(* CODESYS project Estação 2 - Measuring (2022).project

Project tree, tasks and I/O mapping:
  Device : CPX-CEC-C1-V3, Festo AG & Co. KG, order no. 3473128, version 3.5.7.37
      unmapped channels: Rotary switch
    application Application
      libraries: Standard, * (System); CAA CiA 405, 3.5.7.0 (CAA Technical Workgroup)
      task MainTask (cyclic, interval t#20ms, priority 20) calls PLC_PRG
      program PLC_PRG [ST]
      function ATUALIZAR_VALORES [ST]
      visualisation Visualization
      global variables GVL
      function INICIALIZACAO [ST]
      program teste_comunicacao [ST]
    CANbus : CANbus, 3S - Smart Software Solutions GmbH, version 3.5.12.0
        settings: Baudrate = 1000 kbit/s
      CANopen_Manager : CANopen_Manager, 3S - Smart Software Solutions GmbH, version 3.5.10.0
          settings: Sync CycleTime in Microseconds = 8000; Synchronous Window Length = 0; Enable Heartbeat generation = FALSE; Factory Settings Default = FALSE; Expert Settings Default = TRUE; ConfigVersion = 50659584
        CTEU_CO : CTEU-CO, Festo AG & Co. KG, order no. 570038, version 0.3223089.CTEU_CO.3.3
            settings: NODEIDSAVED = 1; SDO Timeout = 1000000; EXPERTSETTINGS = TRUE; PDO 16#1400.COBID = 16#00000201; Process by CANopenManager = TRUE; PDO 16#1401.COBID = 16#00000301; Process by CANopenManager = TRUE; PDO 16#1800.COBID = 16#00000181; Process by CANopenManager = TRUE; PDO 16#1801.COBID = 16#00000281; Process by CANopenManager = TRUE; 8-Bit Digital Output 1-8.Subindex = 16#01; 8-Bit Digital Output 9-16.Subindex = 16#02; 8-Bit Digital Output 17-24.Subindex = 16#03; 8-Bit Digital Output 25-32.Subindex = 16#04; 8-Bit Digital Output 33-40.Subindex = 16#05; 8-Bit Digital Output 41-48.Subindex = 16#06; 8-Bit Digital Output 49-56.Subindex = 16#07; 8-Bit Digital Output 75-64.Subindex = 16#08; 8-Bit Digital Output 65-72.Subindex = 16#09; 8-Bit Digital Output 73-80.Subindex = 16#0A; 8-Bit Digital Output 81-88.Subindex = 16#0B; 8-Bit Digital Output 89-96.Subindex = 16#0C; 8-Bit Digital Output 97-104.Subindex = 16#0D; 8-Bit Digital Output 105-112.Subindex = 16#0E; 8-Bit Digital Output 113-120.Subindex = 16#0F; 8-Bit Digital Input 1-8.Subindex = 16#01; 8-Bit Digital Input 9-16.Subindex = 16#02; 8-Bit Digital Input 17-24.Subindex = 16#03; 8-Bit Digital Input 25-32.Subindex = 16#04; 8-Bit Digital Input 33-40.Subindex = 16#05; 8-Bit Digital Input 41-48.Subindex = 16#06; 8-Bit Digital Input 49-56.Subindex = 16#07; 8-Bit Digital Input 57-64.Subindex = 16#08; 8-Bit Digital Input 65-72.Subindex = 16#09; 8-Bit Digital Input 73-80.Subindex = 16#0A; 8-Bit Digital Input 81-88.Subindex = 16#0B; 8-Bit Digital Input 89-96.Subindex = 16#0C; 8-Bit Digital Input 97-104.Subindex = 16#0D; 8-Bit Digital Input 105-112.Subindex = 16#0E;
              8-Bit Digital Input 113-120.Subindex = 16#0F; SDO List.Set Guardtime.Index = 16#100C; SDO List.Set Guardtime.Subindex = 16#00; SDO List.Set Guardtime.Value = 16#00000000; SDO List.Set Guardtime.Size = 16; SDO List.Set Guardtime.AbortIfError = FALSE; SDO List.Set Guardtime.JumpToLine = FALSE; SDO List.Set Guardtime.Line = 0; SDO List.Set Lifetime.Index = 16#100D; SDO List.Set Lifetime.Subindex = 16#00; SDO List.Set Lifetime.Value = 16#00000000; SDO List.Set Lifetime.Size = 8; SDO List.Set Lifetime.AbortIfError = FALSE; SDO List.Set Lifetime.JumpToLine = FALSE; SDO List.Set Lifetime.Line = 0; SDO List.Set Heartbeat Consumer.Index = 16#1016; SDO List.Set Heartbeat Consumer.Subindex = 16#01; SDO List.Set Heartbeat Consumer.Value = 0; SDO List.Set Heartbeat Consumer.Size = 32; SDO List.Set Heartbeat Consumer.AbortIfError = FALSE; SDO List.Set Heartbeat Consumer.JumpToLine = FALSE; SDO List.Set Heartbeat Consumer.Line = 0; SDO List.Set Heartbeat Consumer.Index = 16#1016; SDO List.Set Heartbeat Consumer.Subindex = 16#02; SDO List.Set Heartbeat Consumer.Value = 0; SDO List.Set Heartbeat Consumer.Size = 32; SDO List.Set Heartbeat Consumer.AbortIfError = FALSE; SDO List.Set Heartbeat Consumer.JumpToLine = FALSE; SDO List.Set Heartbeat Consumer.Line = 0; SDO List.Set Heartbeat Consumer.Index = 16#1016; SDO List.Set Heartbeat Consumer.Subindex = 16#03; SDO List.Set Heartbeat Consumer.Value = 0; SDO List.Set Heartbeat Consumer.Size = 32; SDO List.Set Heartbeat Consumer.AbortIfError = FALSE; SDO List.Set Heartbeat Consumer.JumpToLine = FALSE; SDO List.Set Heartbeat Consumer.Line = 0; SDO List.Set Heartbeat Producer.Index = 16#1017; SDO List.Set Heartbeat Producer.Subindex = 16#00; SDO List.Set Heartbeat Producer.Value = 16#00000000; SDO List.Set Heartbeat Producer.Size = 16;
              SDO List.Set Heartbeat Producer.AbortIfError = FALSE; SDO List.Set Heartbeat Producer.JumpToLine = FALSE; SDO List.Set Heartbeat Producer.Line = 0; SDO List.Disable PDO.Index = 16#1400; SDO List.Disable PDO.Subindex = 16#01; SDO List.Disable PDO.Value = 16#80000201; SDO List.Disable PDO.Size = 32; SDO List.Disable PDO.AbortIfError = FALSE; SDO List.Disable PDO.JumpToLine = FALSE; SDO List.Disable PDO.Line = 0; SDO List.Set transmission type.Index = 16#1400; SDO List.Set transmission type.Subindex = 16#02; SDO List.Set transmission type.Value = 16#FF; SDO List.Set transmission type.Size = 8; SDO List.Set transmission type.AbortIfError = FALSE; SDO List.Set transmission type.JumpToLine = FALSE; SDO List.Set transmission type.Line = 0; SDO List.Clear pdo mapping.Index = 16#1600; SDO List.Clear pdo mapping.Subindex = 16#00; SDO List.Clear pdo mapping.Value = 16#0; SDO List.Clear pdo mapping.Size = 8; SDO List.Clear pdo mapping.AbortIfError = FALSE; SDO List.Clear pdo mapping.JumpToLine = FALSE; SDO List.Clear pdo mapping.Line = 0; SDO List.Set Mapping.Index = 16#1600; SDO List.Set Mapping.Subindex = 16#01; SDO List.Set Mapping.Value = 16#62000108; SDO List.Set Mapping.Size = 32; SDO List.Set Mapping.AbortIfError = FALSE; SDO List.Set Mapping.JumpToLine = FALSE; SDO List.Set Mapping.Line = 0; SDO List.Set Mapping.Index = 16#1600; SDO List.Set Mapping.Subindex = 16#02; SDO List.Set Mapping.Value = 16#62000208; SDO List.Set Mapping.Size = 32; SDO List.Set Mapping.AbortIfError = FALSE; SDO List.Set Mapping.JumpToLine = FALSE; SDO List.Set Mapping.Line = 0; SDO List.Set Mapping.Index = 16#1600; SDO List.Set Mapping.Subindex = 16#03;
              SDO List.Set Mapping.Value = 16#62000308; SDO List.Set Mapping.Size = 32; SDO List.Set Mapping.AbortIfError = FALSE; SDO List.Set Mapping.JumpToLine = FALSE; SDO List.Set Mapping.Line = 0; SDO List.Set Mapping.Index = 16#1600; SDO List.Set Mapping.Subindex = 16#04; SDO List.Set Mapping.Value = 16#62000408; SDO List.Set Mapping.Size = 32; SDO List.Set Mapping.AbortIfError = FALSE; SDO List.Set Mapping.JumpToLine = FALSE; SDO List.Set Mapping.Line = 0; SDO List.Set Mapping.Index = 16#1600; SDO List.Set Mapping.Subindex = 16#05; SDO List.Set Mapping.Value = 16#62000508; SDO List.Set Mapping.Size = 32; SDO List.Set Mapping.AbortIfError = FALSE; SDO List.Set Mapping.JumpToLine = FALSE; SDO List.Set Mapping.Line = 0; SDO List.Set Mapping.Index = 16#1600; SDO List.Set Mapping.Subindex = 16#06; SDO List.Set Mapping.Value = 16#62000608; SDO List.Set Mapping.Size = 32; SDO List.Set Mapping.AbortIfError = FALSE; SDO List.Set Mapping.JumpToLine = FALSE; SDO List.Set Mapping.Line = 0; SDO List.Set Mapping.Index = 16#1600; SDO List.Set Mapping.Subindex = 16#07; SDO List.Set Mapping.Value = 16#62000708; SDO List.Set Mapping.Size = 32; SDO List.Set Mapping.AbortIfError = FALSE; SDO List.Set Mapping.JumpToLine = FALSE; SDO List.Set Mapping.Line = 0; SDO List.Set Mapping.Index = 16#1600; SDO List.Set Mapping.Subindex = 16#08; SDO List.Set Mapping.Value = 16#62000808; SDO List.Set Mapping.Size = 32; SDO List.Set Mapping.AbortIfError = FALSE; SDO List.Set Mapping.JumpToLine = FALSE; SDO List.Set Mapping.Line = 0;
              SDO List.Set number of mappings.Index = 16#1600; SDO List.Set number of mappings.Subindex = 16#00; SDO List.Set number of mappings.Value = 16#08; SDO List.Set number of mappings.Size = 8; SDO List.Set number of mappings.AbortIfError = FALSE; SDO List.Set number of mappings.JumpToLine = FALSE; SDO List.Set number of mappings.Line = 0; SDO List.Set and enable COB-ID.Index = 16#1400; SDO List.Set and enable COB-ID.Subindex = 16#01; SDO List.Set and enable COB-ID.Value = 16#00000201; SDO List.Set and enable COB-ID.Size = 32; SDO List.Set and enable COB-ID.AbortIfError = FALSE; SDO List.Set and enable COB-ID.JumpToLine = FALSE; SDO List.Set and enable COB-ID.Line = 0; SDO List.Disable PDO.Index = 16#1401; SDO List.Disable PDO.Subindex = 16#01; SDO List.Disable PDO.Value = 16#80000301; SDO List.Disable PDO.Size = 32; SDO List.Disable PDO.AbortIfError = FALSE; SDO List.Disable PDO.JumpToLine = FALSE; SDO List.Disable PDO.Line = 0; SDO List.Set transmission type.Index = 16#1401; SDO List.Set transmission type.Subindex = 16#02; SDO List.Set transmission type.Value = 16#FF; SDO List.Set transmission type.Size = 8; SDO List.Set transmission type.AbortIfError = FALSE; SDO List.Set transmission type.JumpToLine = FALSE; SDO List.Set transmission type.Line = 0; SDO List.Clear pdo mapping.Index = 16#1601; SDO List.Clear pdo mapping.Subindex = 16#00; SDO List.Clear pdo mapping.Value = 16#0; SDO List.Clear pdo mapping.Size = 8; SDO List.Clear pdo mapping.AbortIfError = FALSE; SDO List.Clear pdo mapping.JumpToLine = FALSE; SDO List.Clear pdo mapping.Line = 0; SDO List.Set Mapping.Index = 16#1601; SDO List.Set Mapping.Subindex = 16#01; SDO List.Set Mapping.Value = 16#62000908; SDO List.Set Mapping.Size = 32; SDO List.Set Mapping.AbortIfError = FALSE;
              SDO List.Set Mapping.JumpToLine = FALSE; SDO List.Set Mapping.Line = 0; SDO List.Set Mapping.Index = 16#1601; SDO List.Set Mapping.Subindex = 16#02; SDO List.Set Mapping.Value = 16#62000A08; SDO List.Set Mapping.Size = 32; SDO List.Set Mapping.AbortIfError = FALSE; SDO List.Set Mapping.JumpToLine = FALSE; SDO List.Set Mapping.Line = 0; SDO List.Set Mapping.Index = 16#1601; SDO List.Set Mapping.Subindex = 16#03; SDO List.Set Mapping.Value = 16#62000B08; SDO List.Set Mapping.Size = 32; SDO List.Set Mapping.AbortIfError = FALSE; SDO List.Set Mapping.JumpToLine = FALSE; SDO List.Set Mapping.Line = 0; SDO List.Set Mapping.Index = 16#1601; SDO List.Set Mapping.Subindex = 16#04; SDO List.Set Mapping.Value = 16#62000C08; SDO List.Set Mapping.Size = 32; SDO List.Set Mapping.AbortIfError = FALSE; SDO List.Set Mapping.JumpToLine = FALSE; SDO List.Set Mapping.Line = 0; SDO List.Set Mapping.Index = 16#1601; SDO List.Set Mapping.Subindex = 16#05; SDO List.Set Mapping.Value = 16#62000D08; SDO List.Set Mapping.Size = 32; SDO List.Set Mapping.AbortIfError = FALSE; SDO List.Set Mapping.JumpToLine = FALSE; SDO List.Set Mapping.Line = 0; SDO List.Set Mapping.Index = 16#1601; SDO List.Set Mapping.Subindex = 16#06; SDO List.Set Mapping.Value = 16#62000E08; SDO List.Set Mapping.Size = 32; SDO List.Set Mapping.AbortIfError = FALSE; SDO List.Set Mapping.JumpToLine = FALSE; SDO List.Set Mapping.Line = 0; SDO List.Set Mapping.Index = 16#1601; SDO List.Set Mapping.Subindex = 16#07; SDO List.Set Mapping.Value = 16#62000F08;
              SDO List.Set Mapping.Size = 32; SDO List.Set Mapping.AbortIfError = FALSE; SDO List.Set Mapping.JumpToLine = FALSE; SDO List.Set Mapping.Line = 0; SDO List.Set Mapping.Index = 16#1601; SDO List.Set Mapping.Subindex = 16#08; SDO List.Set Mapping.Value = 16#62001008; SDO List.Set Mapping.Size = 32; SDO List.Set Mapping.AbortIfError = FALSE; SDO List.Set Mapping.JumpToLine = FALSE; SDO List.Set Mapping.Line = 0; SDO List.Set number of mappings.Index = 16#1601; SDO List.Set number of mappings.Subindex = 16#00; SDO List.Set number of mappings.Value = 16#08; SDO List.Set number of mappings.Size = 8; SDO List.Set number of mappings.AbortIfError = FALSE; SDO List.Set number of mappings.JumpToLine = FALSE; SDO List.Set number of mappings.Line = 0; SDO List.Set and enable COB-ID.Index = 16#1401; SDO List.Set and enable COB-ID.Subindex = 16#01; SDO List.Set and enable COB-ID.Value = 16#00000301; SDO List.Set and enable COB-ID.Size = 32; SDO List.Set and enable COB-ID.AbortIfError = FALSE; SDO List.Set and enable COB-ID.JumpToLine = FALSE; SDO List.Set and enable COB-ID.Line = 0; SDO List.Disable PDO.Index = 16#1800; SDO List.Disable PDO.Subindex = 16#01; SDO List.Disable PDO.Value = 16#80000181; SDO List.Disable PDO.Size = 32; SDO List.Disable PDO.AbortIfError = FALSE; SDO List.Disable PDO.JumpToLine = FALSE; SDO List.Disable PDO.Line = 0; SDO List.Set transmission type.Index = 16#1800; SDO List.Set transmission type.Subindex = 16#02; SDO List.Set transmission type.Value = 16#FF; SDO List.Set transmission type.Size = 8; SDO List.Set transmission type.AbortIfError = FALSE; SDO List.Set transmission type.JumpToLine = FALSE; SDO List.Set transmission type.Line = 0; SDO List.Set inhibit time.Index = 16#1800;
              SDO List.Set inhibit time.Subindex = 16#03; SDO List.Set inhibit time.Value = 16#0000; SDO List.Set inhibit time.Size = 16; SDO List.Set inhibit time.AbortIfError = FALSE; SDO List.Set inhibit time.JumpToLine = FALSE; SDO List.Set inhibit time.Line = 0; SDO List.Set event time.Index = 16#1800; SDO List.Set event time.Subindex = 16#05; SDO List.Set event time.Value = 16#0000; SDO List.Set event time.Size = 16; SDO List.Set event time.AbortIfError = FALSE; SDO List.Set event time.JumpToLine = FALSE; SDO List.Set event time.Line = 0; SDO List.Clear pdo mapping.Index = 16#1A00; SDO List.Clear pdo mapping.Subindex = 16#00; SDO List.Clear pdo mapping.Value = 16#0; SDO List.Clear pdo mapping.Size = 8; SDO List.Clear pdo mapping.AbortIfError = FALSE; SDO List.Clear pdo mapping.JumpToLine = FALSE; SDO List.Clear pdo mapping.Line = 0; SDO List.Set Mapping.Index = 16#1A00; SDO List.Set Mapping.Subindex = 16#01; SDO List.Set Mapping.Value = 16#60000108; SDO List.Set Mapping.Size = 32; SDO List.Set Mapping.AbortIfError = FALSE; SDO List.Set Mapping.JumpToLine = FALSE; SDO List.Set Mapping.Line = 0; SDO List.Set Mapping.Index = 16#1A00; SDO List.Set Mapping.Subindex = 16#02; SDO List.Set Mapping.Value = 16#60000208; SDO List.Set Mapping.Size = 32; SDO List.Set Mapping.AbortIfError = FALSE; SDO List.Set Mapping.JumpToLine = FALSE; SDO List.Set Mapping.Line = 0; SDO List.Set Mapping.Index = 16#1A00; SDO List.Set Mapping.Subindex = 16#03; SDO List.Set Mapping.Value = 16#60000308; SDO List.Set Mapping.Size = 32; SDO List.Set Mapping.AbortIfError = FALSE; SDO List.Set Mapping.JumpToLine = FALSE;
              SDO List.Set Mapping.Line = 0; SDO List.Set Mapping.Index = 16#1A00; SDO List.Set Mapping.Subindex = 16#04; SDO List.Set Mapping.Value = 16#60000408; SDO List.Set Mapping.Size = 32; SDO List.Set Mapping.AbortIfError = FALSE; SDO List.Set Mapping.JumpToLine = FALSE; SDO List.Set Mapping.Line = 0; SDO List.Set Mapping.Index = 16#1A00; SDO List.Set Mapping.Subindex = 16#05; SDO List.Set Mapping.Value = 16#60000508; SDO List.Set Mapping.Size = 32; SDO List.Set Mapping.AbortIfError = FALSE; SDO List.Set Mapping.JumpToLine = FALSE; SDO List.Set Mapping.Line = 0; SDO List.Set Mapping.Index = 16#1A00; SDO List.Set Mapping.Subindex = 16#06; SDO List.Set Mapping.Value = 16#60000608; SDO List.Set Mapping.Size = 32; SDO List.Set Mapping.AbortIfError = FALSE; SDO List.Set Mapping.JumpToLine = FALSE; SDO List.Set Mapping.Line = 0; SDO List.Set Mapping.Index = 16#1A00; SDO List.Set Mapping.Subindex = 16#07; SDO List.Set Mapping.Value = 16#60000708; SDO List.Set Mapping.Size = 32; SDO List.Set Mapping.AbortIfError = FALSE; SDO List.Set Mapping.JumpToLine = FALSE; SDO List.Set Mapping.Line = 0; SDO List.Set Mapping.Index = 16#1A00; SDO List.Set Mapping.Subindex = 16#08; SDO List.Set Mapping.Value = 16#60000808; SDO List.Set Mapping.Size = 32; SDO List.Set Mapping.AbortIfError = FALSE; SDO List.Set Mapping.JumpToLine = FALSE; SDO List.Set Mapping.Line = 0; SDO List.Set number of mappings.Index = 16#1A00; SDO List.Set number of mappings.Subindex = 16#00; SDO List.Set number of mappings.Value = 16#08; SDO List.Set number of mappings.Size = 8;
              SDO List.Set number of mappings.AbortIfError = FALSE; SDO List.Set number of mappings.JumpToLine = FALSE; SDO List.Set number of mappings.Line = 0; SDO List.Set and enable COB-ID.Index = 16#1800; SDO List.Set and enable COB-ID.Subindex = 16#01; SDO List.Set and enable COB-ID.Value = 16#00000181; SDO List.Set and enable COB-ID.Size = 32; SDO List.Set and enable COB-ID.AbortIfError = FALSE; SDO List.Set and enable COB-ID.JumpToLine = FALSE; SDO List.Set and enable COB-ID.Line = 0; SDO List.Disable PDO.Index = 16#1801; SDO List.Disable PDO.Subindex = 16#01; SDO List.Disable PDO.Value = 16#80000281; SDO List.Disable PDO.Size = 32; SDO List.Disable PDO.AbortIfError = FALSE; SDO List.Disable PDO.JumpToLine = FALSE; SDO List.Disable PDO.Line = 0; SDO List.Set transmission type.Index = 16#1801; SDO List.Set transmission type.Subindex = 16#02; SDO List.Set transmission type.Value = 16#FF; SDO List.Set transmission type.Size = 8; SDO List.Set transmission type.AbortIfError = FALSE; SDO List.Set transmission type.JumpToLine = FALSE; SDO List.Set transmission type.Line = 0; SDO List.Set inhibit time.Index = 16#1801; SDO List.Set inhibit time.Subindex = 16#03; SDO List.Set inhibit time.Value = 16#0000; SDO List.Set inhibit time.Size = 16; SDO List.Set inhibit time.AbortIfError = FALSE; SDO List.Set inhibit time.JumpToLine = FALSE; SDO List.Set inhibit time.Line = 0; SDO List.Set event time.Index = 16#1801; SDO List.Set event time.Subindex = 16#05; SDO List.Set event time.Value = 16#0000; SDO List.Set event time.Size = 16; SDO List.Set event time.AbortIfError = FALSE; SDO List.Set event time.JumpToLine = FALSE; SDO List.Set event time.Line = 0; SDO List.Clear pdo mapping.Index = 16#1A01; SDO List.Clear pdo mapping.Subindex = 16#00;
              SDO List.Clear pdo mapping.Value = 16#0; SDO List.Clear pdo mapping.Size = 8; SDO List.Clear pdo mapping.AbortIfError = FALSE; SDO List.Clear pdo mapping.JumpToLine = FALSE; SDO List.Clear pdo mapping.Line = 0; SDO List.Set Mapping.Index = 16#1A01; SDO List.Set Mapping.Subindex = 16#01; SDO List.Set Mapping.Value = 16#60000908; SDO List.Set Mapping.Size = 32; SDO List.Set Mapping.AbortIfError = FALSE; SDO List.Set Mapping.JumpToLine = FALSE; SDO List.Set Mapping.Line = 0; SDO List.Set Mapping.Index = 16#1A01; SDO List.Set Mapping.Subindex = 16#02; SDO List.Set Mapping.Value = 16#60000A08; SDO List.Set Mapping.Size = 32; SDO List.Set Mapping.AbortIfError = FALSE; SDO List.Set Mapping.JumpToLine = FALSE; SDO List.Set Mapping.Line = 0; SDO List.Set Mapping.Index = 16#1A01; SDO List.Set Mapping.Subindex = 16#03; SDO List.Set Mapping.Value = 16#60000B08; SDO List.Set Mapping.Size = 32; SDO List.Set Mapping.AbortIfError = FALSE; SDO List.Set Mapping.JumpToLine = FALSE; SDO List.Set Mapping.Line = 0; SDO List.Set Mapping.Index = 16#1A01; SDO List.Set Mapping.Subindex = 16#04; SDO List.Set Mapping.Value = 16#60000C08; SDO List.Set Mapping.Size = 32; SDO List.Set Mapping.AbortIfError = FALSE; SDO List.Set Mapping.JumpToLine = FALSE; SDO List.Set Mapping.Line = 0; SDO List.Set Mapping.Index = 16#1A01; SDO List.Set Mapping.Subindex = 16#05; SDO List.Set Mapping.Value = 16#60000D08; SDO List.Set Mapping.Size = 32; SDO List.Set Mapping.AbortIfError = FALSE; SDO List.Set Mapping.JumpToLine = FALSE; SDO List.Set Mapping.Line = 0;
              SDO List.Set Mapping.Index = 16#1A01; SDO List.Set Mapping.Subindex = 16#06; SDO List.Set Mapping.Value = 16#60000E08; SDO List.Set Mapping.Size = 32; SDO List.Set Mapping.AbortIfError = FALSE; SDO List.Set Mapping.JumpToLine = FALSE; SDO List.Set Mapping.Line = 0; SDO List.Set Mapping.Index = 16#1A01; SDO List.Set Mapping.Subindex = 16#07; SDO List.Set Mapping.Value = 16#60000F08; SDO List.Set Mapping.Size = 32; SDO List.Set Mapping.AbortIfError = FALSE; SDO List.Set Mapping.JumpToLine = FALSE; SDO List.Set Mapping.Line = 0; SDO List.Set Mapping.Index = 16#1A01; SDO List.Set Mapping.Subindex = 16#08; SDO List.Set Mapping.Value = 16#60001008; SDO List.Set Mapping.Size = 32; SDO List.Set Mapping.AbortIfError = FALSE; SDO List.Set Mapping.JumpToLine = FALSE; SDO List.Set Mapping.Line = 0; SDO List.Set number of mappings.Index = 16#1A01; SDO List.Set number of mappings.Subindex = 16#00; SDO List.Set number of mappings.Value = 16#08; SDO List.Set number of mappings.Size = 8; SDO List.Set number of mappings.AbortIfError = FALSE; SDO List.Set number of mappings.JumpToLine = FALSE; SDO List.Set number of mappings.Line = 0; SDO List.Set and enable COB-ID.Index = 16#1801; SDO List.Set and enable COB-ID.Subindex = 16#01; SDO List.Set and enable COB-ID.Value = 16#00000281; SDO List.Set and enable COB-ID.Size = 32; SDO List.Set and enable COB-ID.AbortIfError = FALSE; SDO List.Set and enable COB-ID.JumpToLine = FALSE; SDO List.Set and enable COB-ID.Line = 0; ConfigVersion = 50659584
            unmapped channels: 8-Bit Digital Output 1-8, 8-Bit Digital Output 9-16, 8-Bit Digital Output 17-24, 8-Bit Digital Output 25-32, 8-Bit Digital Output 33-40, 8-Bit Digital Output 41-48, 8-Bit Digital Output 49-56, 8-Bit Digital Output 75-64, 8-Bit Digital Output 65-72, 8-Bit Digital Output 73-80, 8-Bit Digital Output 81-88, 8-Bit Digital Output 89-96, 8-Bit Digital Output 97-104, 8-Bit Digital Output 105-112, 8-Bit Digital Output 113-120, 8-Bit Digital Output 121-128, 8-Bit Digital Input 1-8, 8-Bit Digital Input 9-16, 8-Bit Digital Input 17-24, 8-Bit Digital Input 25-32, 8-Bit Digital Input 33-40, 8-Bit Digital Input 41-48, 8-Bit Digital Input 49-56, 8-Bit Digital Input 57-64, 8-Bit Digital Input 65-72, 8-Bit Digital Input 73-80, 8-Bit Digital Input 81-88, 8-Bit Digital Input 89-96, 8-Bit Digital Input 97-104, 8-Bit Digital Input 105-112, 8-Bit Digital Input 113-120, 8-Bit Digital Input 121-128
    Ethernet : Ethernet, 3S - Smart Software Solutions GmbH, version 3.5.10.0
        settings: IPAddress = [192,168,2,30]; SubnetMask = [255,255,0,0]; GatewayAddress = [192,168,1,1]; MACAddress = [16#00,16#0E,16#F0,16#5D,16#13,16#D4]; NetworkInterfaceName = 'eth0'; NetworkInterfaceName = "eth0"; SaveCommunicationSettings = FALSE
      ModbusTCP_Slave_Device : ModbusTCP Slave Device, 3S - Smart Software Solutions GmbH, version 3.5.10.0
          unmapped channels: Inputs, Outputs
    PLC_Diagnosis : PLC-Diagnosis, Festo AG & Co. KG, version 3.5.4.1
    CPX_System : CPX_System, Festo AG & Co. KG, order no. 3473128, version 1.258
      _8DI_8DO_1 : 8DI/8DO, Festo AG & Co. KG, order no. 526257, version 1.258
          settings:  = 0;  = 1;  = 1;  = 1;  = 1;  = 0;  = 1;  = 1;  = 0;  = 0;  = 0;  = 0;  = 0;  = 0;  = 0;  = 0;  = 0;  = 0;  = 0;  = 0;  = 0;  = 0;  = 0;  = 0;  = 0;  = 0;  = 0;  = 0;  = 0;  = 0;  = 0;  = 0;  = 0;  = 0;  = 0;  = 0;  = 0;  = 0;  = 0;  = 0;
             = 0;  = 0;  = 0;  = 0;  = 0;  = 0;  = 0;  = 0;  = 0;  = 0;  = 0;  = 0;  = 0;  = 0;  = 0;  = 0;  = 0;  = 0;  = 0;  = 0;  = 0;  = 0;  = 0;  = 0;  = 0;  = 0;  = 0;  = 0;  = 0;  = 0;  = 0;  = 0;  = 0;  = 0;  = 0;  = 0;  = 0;  = 0;  = 0;  = 0;
             = 576751027668385792;  = 'PI%i.0.0.1=1';  = 'PI%i.0.1.1=1';  = 'PI%i.0.2.1=1';  = 'PI%i.1.0.1=1';  = 'PI%i.1.1.1=0';  = 'PI%i.1.4.2=1';  = 'PI%i.1.6.2=1';  = 'PI%i.6.0.1=0';  = 'PI%i.6.1.1=0';  = 'PI%i.6.2.1=0';  = 'PI%i.6.3.1=0';  = 'PI%i.6.4.1=0';  = 'PI%i.6.5.1=0';  = 'PI%i.6.6.1=0';  = 'PI%i.6.7.1=0';  = dd39f1e1;  = 6
          unmapped channels: Input 0, Output 0
      _8DI_8DO : 8DI/8DO, Festo AG & Co. KG, order no. 526257, version 1.258
          settings:  = 0;  = 1;  = 1;  = 1;  = 1;  = 0;  = 1;  = 1;  = 0;  = 0;  = 0;  = 0;  = 0;  = 0;  = 0;  = 0;  = 0;  = 0;  = 0;  = 0;  = 0;  = 0;  = 0;  = 0;  = 0;  = 0;  = 0;  = 0;  = 0;  = 0;  = 0;  = 0;  = 0;  = 0;  = 0;  = 0;  = 0;  = 0;  = 0;  = 0;
             = 0;  = 0;  = 0;  = 0;  = 0;  = 0;  = 0;  = 0;  = 0;  = 0;  = 0;  = 0;  = 0;  = 0;  = 0;  = 0;  = 0;  = 0;  = 0;  = 0;  = 0;  = 0;  = 0;  = 0;  = 0;  = 0;  = 0;  = 0;  = 0;  = 0;  = 0;  = 0;  = 0;  = 0;  = 0;  = 0;  = 0;  = 0;  = 0;  = 0;
             = 576751027668385792;  = 'PI%i.0.0.1=1';  = 'PI%i.0.1.1=1';  = 'PI%i.0.2.1=1';  = 'PI%i.1.0.1=1';  = 'PI%i.1.1.1=0';  = 'PI%i.1.4.2=1';  = 'PI%i.1.6.2=1';  = 'PI%i.6.0.1=0';  = 'PI%i.6.1.1=0';  = 'PI%i.6.2.1=0';  = 'PI%i.6.3.1=0';  = 'PI%i.6.4.1=0';  = 'PI%i.6.5.1=0';  = 'PI%i.6.6.1=0';  = 'PI%i.6.7.1=0';  = dd4a6dfc;  = 6
          unmapped channels: Input 0, Output 0
      CEC_C1_V3 : CEC-C1-V3, Festo AG & Co. KG, order no. 3473128, version 1.258
          settings:  = 0;  = 233179645480448;  = 503490752;  = 65535;  = 16885952;  = 13959208;  = 1f5d13d4;  = 5
  text list GlobalTextList
*)

// Device/Application/GVL
{attribute 'qualified_only'}
VAR_GLOBAL
//Entradas
	//Sensores
	S_inicio 		AT %IX1.0 :BOOL; //Sensor de inicio da esteira
	S_meio 	 		AT %IX1.1 :BOOL; //Sensor do meio da esteira
	S_fim_ramp		AT %IX1.2 :BOOL; //Sensor do fim da esteira / rampa de descarte
	S_dist_digit    AT %IX1.3 :BOOL; //Sinal digital do sensor de distância
	S_G_aberta 		AT %IX1.4  :BOOL; //Garra aberta
	S_G_cima	    AT %IX1.5 :BOOL; //Cilindro avançado para baixo
	S_G_esteira  	AT %IX1.6  :BOOL; //Modulo de giro na posição da esteira
	S_G_camera  	AT %IX1.7  :BOOL; //Modulo de giro na posição da camera
	
	//IHM
	Start_btn 		AT	%IX2.0	:BOOL;  //Botão de start
	Stop_btn 		AT	%IX2.1	:BOOL;	//Botão de stop (NF)
	Chave 			AT	%IX2.2	:BOOL;	//Chave auto/manual
	Reset_btn 		AT	%IX2.3	:BOOL;	//Botão de reset
	I4_IHM			AT	%IX2.4	:BOOL;	//Bit de saída 4 da IHM
	I5_IHM			AT	%IX2.5	:BOOL;	//Bit de saída 5 da IHM
	I6_IHM 			AT	%IX2.6	:BOOL;	//Bit de saída 6 da IHM
	I7_IHM			AT	%IX2.7	:BOOL;	//Bit de saída 7 da IHM

//Saídas
	//Atuadorres 			
	Esteira_frente 	AT	%QX0.0	:BOOL;	//Mover a esteira para frente
	Esteira_tras 	AT	%QX0.1	:BOOL;	//Mover a esteira para tras
	Separador 	 	AT	%QX0.2	:BOOL;	//Atuar separador
	Stopper		 	AT	%QX0.3	:BOOL;	//Atuar stopper
	Abrir_garra     AT	%QX0.4	:BOOL;	//Abrir a garra
	Descer_garra	AT	%QX0.5	:BOOL;	//Descer a garra
	Mov_giro_cam	AT	%QX0.6	:BOOL;	//Girar a garra para a posição da camera
	//	     		AT	%QX0.7	:BOOL;	
	
	//IHM				
	Start_LED		AT	%QX1.0	:BOOL;	//LED do botão de start
	Reset_LED 		AT	%QX1.1	:BOOL;	//LED do botão de reset
	Q1_LED 			AT	%QX1.2	:BOOL;	//LED sinalizador Q1
	Q2_LED			AT	%QX1.3	:BOOL;	//LED sinalizador Q2
	Q4_IHM			AT	%QX1.4	:BOOL;	//Saída Q4 IHM
	Q5_IHM			AT	%QX1.5	:BOOL;	//Saída Q5 IHM
	Q6_IHM			AT	%QX1.6	:BOOL;	//Saída Q6 IHM
	Q7_IHM 			AT	%QX1.7	:BOOL;	//Saída Q7 IHM
	
//MODBUS bits
	//Entradas
	Mod_I_0_0 		AT %IX20.0 : BOOL; //Iniciar a estação
	Mod_I_0_1	 	AT %IX20.1 : BOOL; //Parar a estação
	Mod_I_0_2 		AT %IX20.2 : BOOL; //Reiniciar a estação 
	Mod_I_0_3 		AT %IX20.3 : BOOL; //Modo entrada (Desativado para essa estação)
	Mod_I_0_4 		AT %IX20.4 : BOOL; //Modo saída (Desativado para essa estação)
	Mod_I_0_5 		AT %IX20.5 : BOOL; //Teste de resposta da estação - IN
	Mod_I_0_6 		AT %IX20.6 : BOOL; 
	Mod_I_0_7 		AT %IX20.7 : BOOL;
	Mod_I_1_0 		AT %IX21.0 : BOOL;
	Mod_I_1_1 		AT %IX21.1 : BOOL;
	Mod_I_1_2 		AT %IX21.2 : BOOL;
	Mod_I_1_3 		AT %IX21.3 : BOOL;
	Mod_I_1_4 		AT %IX21.4 : BOOL;
	Mod_I_1_5	 	AT %IX21.5 : BOOL;
	Mod_I_1_6 		AT %IX21.6 : BOOL;
	Mod_I_1_7 		AT %IX21.7 : BOOL;
	
	//Saídas
	Mod_Q_0_0 		AT %QX18.0 : BOOL; //Estaão em processo
	Mod_Q_0_1	 	AT %QX18.1 : BOOL; //Estação parada
	Mod_Q_0_2 		AT %QX18.2 : BOOL; //Estação aguardando peça
	Mod_Q_0_3 		AT %QX18.3 : BOOL; //Estação em modo entrada (DESATIVADO PARA ESSA ESTAÇÃO)
	Mod_Q_0_4 		AT %QX18.4 : BOOL; //Estação em modo saída (DESATIVADO PARA ESSA ESTAÇÃO)
	Mod_Q_0_5 		AT %QX18.5 : BOOL; //Teste de resposta da estação - OUT
	Mod_Q_0_6 		AT %QX18.6 : BOOL; 
	Mod_Q_0_7 		AT %QX18.7 : BOOL; 
	Mod_Q_1_0 		AT %QX19.0 : BOOL;
	Mod_Q_1_1 		AT %QX19.1 : BOOL; 
	Mod_Q_1_2 		AT %QX19.2 : BOOL;
	Mod_Q_1_3 		AT %QX19.3 : BOOL; 
	Mod_Q_1_4 		AT %QX19.4 : BOOL; 
	Mod_Q_1_5	 	AT %QX19.5 : BOOL;
	Mod_Q_1_6 		AT %QX19.6 : BOOL; 
	Mod_Q_1_7 		AT %QX19.7 : BOOL; 


	
//CANbus BITs - Camera
	camera_In_0 AT %IX3.0 : BOOL; //Tirar foto
	camera_In_1 AT %IX3.1 : BOOL;
	camera_In_2 AT %IX3.2 : BOOL;
	camera_In_3 AT %IX3.3 : BOOL;
	camera_In_4 AT %IX3.4 : BOOL;
	camera_In_5 AT %IX3.5 : BOOL;
	camera_In_6 AT %IX3.6 : BOOL;
	camera_In_7 AT %IX3.7 : BOOL;
	
	camera_out_0 AT %QX2.0 : BOOL; //Resposta da camera
	camera_out_1 AT %QX2.1 : BOOL;
	camera_out_2 AT %QX2.2 : BOOL;
	camera_out_3 AT %QX2.3 : BOOL;
	camera_out_4 AT %QX2.4 : BOOL;
	camera_out_5 AT %QX2.5 : BOOL;
	camera_out_6 AT %QX2.6 : BOOL;
	camera_out_7 AT %QX2.7 : BOOL;

//Sensor de distancia

//Distancia AT  : ;

//Variáveis de lógica
	principal: BOOL;
	processo : BOOL;
	parada : BOOL;
	passo1: BOOL;	
	passo2: BOOL;
	passo3: BOOL;
	passo4: BOOL;
	passo5: BOOL;
	passo6: BOOL;
	passo7: BOOL;
	passo8: BOOL;
	passo9: BOOL;
	passo10: BOOL;
	passo11: BOOL;
	passo12: BOOL;
	passo13: BOOL;
	passo14: BOOL;
	passo15: BOOL;
	passo16: BOOL;
	passo17: BOOL;
	passo18: BOOL;
	passo19: BOOL;
	passo20: BOOL;
	
	start: BOOL; //Start geral
	stop: BOOL;  //Stop geral
	reset: BOOL; //Reset geral
	key: BOOL; //key geral
	
	TON_3: BOOL;
	TON_4: BOOL;
	
	passoR1 :BOOL;
	passoR2 :BOOL;
	passoR3 :BOOL;
	passoR4 :BOOL;
	passoR5 :BOOL;
	passoR6 :BOOL;




END_VAR

// Device/Application/PLC_PRG
PROGRAM PLC_PRG
VAR
TONInst: Standard.TON;
	VarBOOL1: BOOL;
	IN: INT;
	PT: TIME;
	VarBOOL2: BOOL;
	TONInst2: TON;
	TON_2: BOOL;
	TON_1: BOOL;
	
	TONInst3: Ton;
	TONInst4: Ton;
	G_Pronta : BOOL;
	R_Pronto : BOOL;
	
	TONInst5: Ton;
	TON_5: BOOL;
	Cont : INT;
	TON_6: BOOL;
	TONInst6: Ton;
END_VAR

ATUALIZAR_VALORES();
INICIALIZACAO();
teste_comunicacao();

TONInst(IN := TON_1, PT:= T#0.6S);
TONInst2(IN := TON_2, PT:= T#1.3S);
TONInst3(IN := GVL.TON_3, PT:= T#0.2S);
TONInst4(IN := GVL.TON_4, PT:= T#0.2S);
TONInst5(IN := TON_5, PT:= T#0.1S);
TONInst6(IN := TON_6, PT:= T#0.5S);
//VarBOOL2 := TONInst.Q;


IF GVL.start  AND NOT GVL.parada AND NOT GVL.principal THEN 
	GVL.principal := TRUE;
	GVL.Q1_LED := TRUE;
	GVL.Start_LED := FALSE;
	
	GVL.passoR1 := TRUE;
END_IF

IF  GVL.stop THEN
	gvl.processo := FALSE;
	GVL.principal := FALSE;
	GVL.parada := TRUE;
	GVL.Esteira_frente :=FALSE;
	GVL.Esteira_tras :=FALSE;
	GVL.Start_LED := FALSE;
	GVL.Reset_LED := TRUE;
	GVL.Q2_LED := FALSE;
	GVL.Q1_LED := FALSE;
	GVL.TON_3 := FALSE;
	GVL.Q4_IHM := FALSE;
	
END_IF

IF GVL.reset AND NOT GVL.principal AND GVL.parada
THEN
	gvl.processo := FALSE;
	GVL.passo1:= FALSE;
	GVL.passo2:= FALSE;
	GVL.passo3:= FALSE;
	GVL.passo4:= FALSE;
	GVL.passo5:= FALSE;
	GVL.passo6:= FALSE;
	GVL.passo7:= FALSE;
	GVL.passo8:= FALSE;
	GVL.passo9:= FALSE;
	GVL.passo10:= FALSE;
	GVL.passo11:= FALSE;
	GVL.passo12 := FALSE;
	GVL.passo13:= FALSE;
	GVL.passo14:= FALSE;
	GVL.passo15:= FALSE;
	GVL.passo16:= FALSE;
	GVL.passo17:= FALSE;
	GVL.passo18:= FALSE;
	GVL.passo19:= FALSE;
	GVL.passo20:= FALSE;
	
	GVL.Separador:= FALSE;
	GVL.Esteira_frente :=FALSE;
	GVL.Esteira_tras :=FALSE;
	GVL.Stopper := FALSE;
	
	GVL.Abrir_garra := TRUE;
	GVL.Descer_garra := FALSE;
	GVL.Mov_giro_cam := FALSE;
	
	GVL.parada := FALSE;
	TON_1 := FALSE;
	TON_2 := FALSE;
	GVL.TON_3 := FALSE;
	GVL.TON_4 := FALSE;
	GVL.Reset_LED := FALSE;
	
END_IF

IF NOT GVL.principal AND NOT GVL.parada  THEN 
	GVL.Start_LED := TRUE;
END_IF

//IF NOT G_Pronta AND R_Pronto THEN
//	GVL.stop := TRUE;
//END_IF
	

IF GVL.principal AND NOT GVL.parada THEN  //Pisca pisca
	IF TONInst4.Q THEN
		GVL.TON_4 := FALSE;
		GVL.TON_3 := TRUE;
		GVL.Q2_LED := FALSE;
	END_IF
	IF TONInst3.Q THEN
		GVL.TON_3 := FALSE;
		GVL.TON_4 := TRUE;
		GVL.Q2_LED := TRUE;
	END_IF
END_IF

IF GVL.passo1 AND GVL.S_inicio AND NOT GVL.parada THEN
	GVL.passo1 := FALSE;
	GVL.passo2 := TRUE;
	GVL.Q4_IHM := FALSE;
	GVL.Esteira_frente	:= TRUE;
	GVL.TON_3 := TRUE;
	gvl.processo := TRUE;
END_IF

IF GVL.passo2 AND GVL.S_meio AND NOT GVL.parada  THEN
	GVL.passo2 := FALSE;
	GVL.passo3 := TRUE;
	TON_1 := TRUE;	
END_IF

IF GVL.passo3 AND TONInst.Q AND NOT GVL.parada  THEN
	GVL.passo3:= FALSE;
	GVL.passo4:= TRUE;
	TON_1 := FALSE;
	GVL.Esteira_frente := FALSE;
END_IF

IF GVL.passo4 AND NOT GVL.parada  THEN
	GVL.passo4 := FALSE;
	GVL.passo5 := TRUE;
	GVL.Descer_garra := TRUE;
	TON_2 := TRUE;
END_IF

IF GVL.passo5 AND TONInst2.Q AND NOT GVL.parada  THEN
	GVL.passo5 := FALSE;
	GVL.passo6 := TRUE;
	TON_2 := FALSE;
	GVL.Abrir_garra := FALSE;
END_IF

IF GVL.passo6 AND NOT GVL.S_G_aberta AND NOT GVL.parada  THEN
	GVL.passo6 := FALSE;
	GVL.passo7 := TRUE;
	GVL.Descer_garra := FALSE;
END_IF
IF GVL.passo7 AND GVL.S_G_cima AND NOT GVL.parada  THEN
	GVL.passo7:= FALSE;
	GVL.passo8 := TRUE;
	GVL.Mov_giro_cam := TRUE;
END_IF

IF GVL.passo8 AND GVL.S_G_camera AND NOT GVL.parada  THEN
	GVL.passo8 := FALSE;
	GVL.passo9 := TRUE;
	GVL.Descer_garra := TRUE;
	TON_1 := TRUE;
	GVL.camera_out_1 := FALSE;
	GVL.camera_out_2 := FALSE;
	Cont := 0;
END_IF

IF GVL.passo9 AND TONInst.Q AND NOT GVL.parada  THEN
	GVL.passo9 := FALSE;
	GVL.passo10 := TRUE;
	TON_1 := FALSE;
	gvl.camera_out_0 := TRUE;
	TON_5 := TRUE;
	
	
END_IF

IF GVL.passo10 AND TONInst5.Q AND NOT GVL.parada  THEN
	GVL.passo10 := FALSE;
	GVL.passo11 := TRUE;
	TON_5 := FALSE;
	TON_6 := TRUE;
	gvl.camera_out_0 := FALSE;
	
END_IF

IF GVL.passo11  AND GVL.camera_In_3 AND TONInst6.q AND NOT GVL.parada  THEN
	GVL.passo11 := FALSE;
	TON_6 := FALSE;
	Cont := Cont+1;
	
	IF NOT GVL.camera_In_0 AND cont < 3 THEN
	GVL.passo9 := TRUE;
	TON_1 := TRUE;
		IF Cont = 1 THEN
			GVL.camera_out_1 := TRUE;
		END_IF
		IF Cont = 2 THEN
			GVL.camera_out_2 := TRUE;
		END_IF
		gvl.camera_out_0 := FALSE;
	
	END_IF
	
	IF Cont = 3 OR GVL.camera_In_0 THEN
	GVL.passo12 := TRUE;
	GVL.Descer_garra := FALSE;
	END_IF
END_IF

IF GVL.passo12 AND GVL.S_G_cima AND NOT GVL.parada  THEN
	GVL.passo12 := FALSE;
	GVL.passo13 := TRUE;
	GVL.Mov_giro_cam := FALSE;
END_IF

IF GVL.passo13 AND GVL.S_G_esteira  AND NOT GVL.parada THEN
	GVL.passo13 := FALSE;
	GVL.passo14 := TRUE;
	GVL.Descer_garra := TRUE;
	ton_1 := TRUE;
END_IF

IF GVL.passo14 AND TONInst.Q  AND NOT GVL.parada THEN
	GVL.passo14 := FALSE;
	GVL.passo15 := TRUE;
	TON_1 := FALSE;
	GVL.Abrir_garra := TRUE;
END_IF

IF GVL.passo15 AND GVL.S_G_aberta AND NOT GVL.parada  THEN
	GVL.passo15 := FALSE;
	GVL.passo16 := TRUE;
	GVL.Descer_garra := FALSE;
END_IF

IF GVL.passo16 AND GVL.S_G_cima AND NOT GVL.parada  THEN
	GVL.passo16 := FALSE;
	GVL.passo17 := TRUE;
	GVL.Stopper := TRUE;
	GVL.Esteira_frente := TRUE;
	IF GVL.camera_In_0 THEN
		GVL.Separador := FALSE;
		ELSE
		GVL.Separador := TRUE;
	END_IF
END_IF

IF GVL.passo17 AND NOT GVL.S_fim_ramp AND NOT GVL.camera_In_0 AND NOT GVL.parada  THEN
	GVL.passo17 := FALSE;
	GVL.passo19 := TRUE;
	TON_2 := TRUE;
	GVL.Stopper := FALSE;
END_IF

IF GVL.passo17 AND NOT GVL.S_fim_ramp AND GVL.camera_In_0 AND NOT GVL.parada   THEN
	GVL.passo17 := FALSE;
	GVL.passo18 := TRUE;
	GVL.Esteira_frente := FALSE;
	GVL.Stopper := FALSE;
END_IF

IF GVL.passo18 AND GVL.I6_IHM AND NOT GVL.parada THEN
	GVL.passo18 := FALSE;
	GVL.passo19 := TRUE;
	GVL.Esteira_frente := TRUE;
	TON_2 := TRUE;
END_IF


IF GVL.passo19 AND TONInst2.Q AND NOT GVL.parada  THEN
	GVL.passo19 := FALSE;
	GVL.passo1 := TRUE;
	TON_2 := FALSE;
	GVL.Esteira_frente := FALSE;
	GVL.TON_3 := FALSE;
	GVL.TON_4 := FALSE;
	gvl.processo := FALSE;
	GVL.Separador := FALSE;
	GVL.Q4_IHM := TRUE;
	GVL.Q2_LED := FALSE;
END_IF

END_PROGRAM

// Device/Application/ATUALIZAR_VALORES
FUNCTION ATUALIZAR_VALORES : INT
VAR
END_VAR

GVL.Mod_Q_0_0 := GVL.principal;
GVL.Mod_Q_0_1 := GVL.parada;
GVL.Mod_Q_0_2 := GVL.processo;


IF GVL.Start_btn OR GVL.Mod_I_0_0 THEN  //Atualização do valor da variável de start
	GVL.start := TRUE;
	ELSE
	GVL.start := FALSE;
END_IF

IF NOT GVL.Stop_btn OR GVL.Mod_I_0_1 THEN //Atualização do valor da variável de stop
	GVL.stop := TRUE;
	ELSE
	GVL.stop := FALSE;
END_IF

IF GVL.Reset_btn OR GVL.Mod_I_0_2 THEN //Atualização do valor da variável de reset
	GVL.reset := TRUE;
	ELSE
	GVL.reset := FALSE;	
END_IF

IF GVL.Chave OR GVL.Mod_I_0_3 THEN //Atualização do valor da variável da chave
	GVL.key := TRUE;
	ELSE
	GVL.key := FALSE;
END_IF

END_FUNCTION

// Device/Application/INICIALIZACAO
FUNCTION INICIALIZACAO : INT
VAR
	
END_VAR

IF GVL.passoR1 THEN
	GVL.passoR1 := FALSE;
	GVL.passoR2 := TRUE;
	GVL.Abrir_garra := TRUE;
END_IF

IF GVL.passoR2 AND GVL.S_G_aberta THEN
	GVL.passoR2 := FALSE;
	GVL.passoR3 := TRUE;
	GVL.Descer_garra := TRUE;
END_IF

IF GVL.passoR3 AND NOT GVL.S_G_cima THEN
	GVL.passoR3 := FALSE;
	GVL.passoR4 := TRUE;
	GVL.Descer_garra := FALSE;
END_IF

IF GVL.passoR4 AND  GVL.S_G_cima THEN
	GVL.passoR4 := FALSE;
	GVL.passoR5 := TRUE;
	GVL.Mov_giro_cam := TRUE;
END_IF

IF GVL.passoR5 AND NOT GVL.S_G_esteira THEN
	GVL.passoR5 := FALSE;
	GVL.passoR6 := TRUE;
	GVL.Mov_giro_cam := FALSE;
	GVL.passo1 := TRUE;
	GVL.Q4_IHM := TRUE;
END_IF

END_FUNCTION

// Device/Application/teste_comunicacao
PROGRAM teste_comunicacao
VAR
	
	TON_temp_1: TON;
	TON_1: BOOL;	

END_VAR

gvl.Mod_Q_0_5 := gvl.Mod_I_0_5;

END_PROGRAM

// Device/Application/Visualization
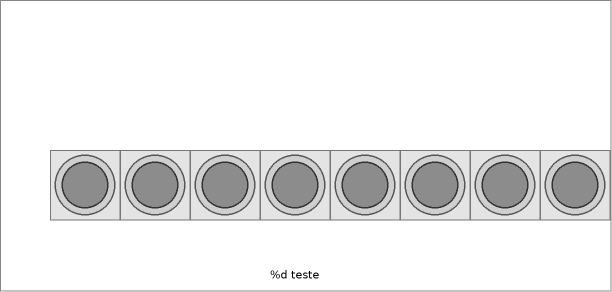
VISUALIZATION Visualization  // 612x292
    PushSwitch (50,150 70x70), variable: GVL.camera_out_0, behaviour: TAP, style: Switch-PushSwitch-Gray
    PushSwitch (120,150 70x70), variable: GVL.camera_out_1, behaviour: TOGGLE, style: Switch-PushSwitch-Gray
    PushSwitch (190,150 70x70), variable: GVL.camera_out_2, behaviour: TOGGLE, style: Switch-PushSwitch-Gray
    PushSwitch (260,150 70x70), variable: GVL.camera_out_3, behaviour: TAP, style: Switch-PushSwitch-Gray
    PushSwitch (330,150 70x70), variable: GVL.camera_out_4, behaviour: TAP, style: Switch-PushSwitch-Gray
    PushSwitch (400,150 70x70), variable: GVL.camera_out_5, behaviour: TAP, style: Switch-PushSwitch-Gray
    PushSwitch (470,150 70x70), variable: GVL.camera_out_6, behaviour: TAP, style: Switch-PushSwitch-Gray
    PushSwitch (540,150 70x70), variable: GVL.camera_out_7, behaviour: TAP, style: Switch-PushSwitch-Gray
    Label (220,260 150x30), "%d teste", invisible if: GVL.Distancia
END_VISUALIZATION
